TYPE ST_TurntablePositionConfig :
STRUCT
    fPosition0 : LREAL;
    fPosition180 : LREAL;
END_STRUCT
END_TYPE

(* stored: Version 1.1.0.1, ProductVersion 3.1.4026.20
   DUT ST_TurntablePositionConfig: Id {33202455-10a8-459c-be32-744f3e124ef6} *)
